INTERFACE ITF_AxisBase

METHOD Disable
END_METHOD

METHOD Enable : BOOL
END_METHOD

PROPERTY Enabled : BOOL
GET
END_GET
END_PROPERTY

PROPERTY EnableNegativeDirection : bool
GET
END_GET
SET
END_SET
END_PROPERTY

PROPERTY Override : lreal
GET
END_GET
SET
END_SET
END_PROPERTY

METHOD Reset
END_METHOD

PROPERTY SafetyOk : BOOL
GET
END_GET
SET
END_SET
END_PROPERTY

PROPERTY Status : REFERENCE TO ST_AxisStatus
GET
END_GET
END_PROPERTY

END_INTERFACE

(* stored: Version 1.1.0.1, ProductVersion 3.1.4024.4
   Itf ITF_AxisBase: Id {7c0b5f35-6961-401c-a129-c286a521a6d4}
   Method Disable: Id {841ea02a-a785-4841-af47-9ea4c09af8f2}
   Method Enable: Id {4f565508-8f93-4c28-901f-5eaf0c6c6987}
   Property Enabled: Id {6038fc20-3e04-4c2e-9804-b028908d58a3}
   Get Get: Id {09ee6104-6e42-48f9-86a9-c740d6ac4e0c}
   Property EnableNegativeDirection: Id {79b8ffa5-86f4-46fa-8e6d-3ee24842e46f}
   Get Get: Id {a6662a0e-841e-4315-9bf0-606c3c29810f}
   Set Set: Id {a0270660-c8a3-45a3-9d33-1cdbb5fae15c}
   Property Override: Id {279d333c-cb93-4282-b275-6bc17aa72e2b}
   Get Get: Id {07367dfe-a7a1-485e-9ced-ce128cae3c11}
   Set Set: Id {63842dd0-fbce-45b5-89a8-d3c548a80219}
   Method Reset: Id {171c9372-db41-483a-a539-db6009a86252}
   Property SafetyOk: Id {8f92f976-7aad-485b-bda9-4d7a6edf5cfd}
   Get Get: Id {53e675bf-b1aa-48c3-9722-87d0ac1a9d60}
   Set Set: Id {94bca364-204b-4f44-940d-120a68650f06}
   Property Status: Id {717b381b-fd43-4de9-8e91-379e6ed665bb}
   Get Get: Id {859f5a5a-3bbd-4c4b-8847-ba54a2e88d40} *)
